{attribute 'qualified_only'}
{attribute 'strict'}
{attribute 'to_string'}
TYPE DUT_OutputType :
(
	Digital := 0,
	Pwm := 1
);
END_TYPE

(* stored: Version 1.1.0.1
   EnumerationTextList DUT_OutputType: Id {a34b11eb-e2af-482c-aa2e-a29191fc1dc3} *)
